// TIA Portal V17 export
// export: Created 2024-03-30T11:15:04.1625877Z, ExportSetting WithDefaults, DisplayName Totally Integrated Automation Portal, DisplayVersion V17, DisplayName TIA Portal Openness, DisplayVersion V17, DisplayName TIA Portal Version Control Interface, DisplayVersion V17, DisplayName STEP 7 Professional, DisplayVersion V17, DisplayName STEP 7 Safety, DisplayVersion V17, DisplayName WinCC Advanced, DisplayVersion V17
TYPE "typ_VGR"
// stored: IsFailsafeCompliant false
   STRUCT
      x_Start_Park_Position : Bool;
      x_Park_Position_Reached : Bool;
      x_NFC_Start_First : Bool;
      x_NFC_Start : Bool;
      x_NFC_Completed : Bool;
      x_HBW_Storage : Bool;
      x_HBW_Outsource : Bool;
      s_HBW_Outsource_Typ : String;
      x_HBW_Discards : Bool;
      x_HBW_PickedUp : Bool;
      x_MPO_Req_Discard : Bool;
      x_MPO_Discards : Bool;
      x_Ready_For_Outsource : Bool;
      x_State_Process : Bool;
      x_Workpiece_NiO : Bool;
      horizontal_Axis : "typ_Axis";
      vertical_Axis : "typ_Axis";
      rotate_Axis : "typ_Axis";
      Workpiece : "typ_Workpiece";
      Worpiece_Parameters { S7_SetPoint := 'True'} : "typ_Workpiece_Parameters";
      History { S7_SetPoint := 'True'} : Array[1..20] of "typ_History";
      di_Pos_DSI_horizontal : DInt;
      di_Pos_DSI_Collect_vertical : DInt;
      di_Pos_DSI_Discard_vertical : DInt;
      di_Offset_Pos_DSI_NFC_vertical : DInt;
      di_Pos_DSI_rotate : DInt;
      di_Pos_DSO_horizontal : DInt;
      di_Pos_DSO_Collect_vertical : DInt;
      di_Pos_DSO_Discard_vertical : DInt;
      di_Offset_Pos_DSO_vertical : DInt;
      di_Pos_DSO_rotate : DInt;
      di_Pos_Color_horizontal : DInt;
      di_Pos_Color_vertical : DInt;
      di_Pos_Color_rotate : DInt;
      di_Pos_NFC_horizontal : DInt;
      di_Pos_NFC_vertical : DInt;
      di_Pos_NFC_rotate : DInt;
      di_Pos_MPO_horizontal : DInt;
      di_Pos_MPO_vertical : DInt;
      di_Offset_Pos_MPO_vertical : DInt;
      di_Pos_MPO_rotate : DInt;
      di_Pos_Free_MPO_Min_rotate : DInt;
      di_Pos_Free_MPO_Max_rotate : DInt;
      di_Pos_Free_MPO_horizontal : DInt;
      di_Pos_HBW_horizontal : DInt;
      di_Offset_Pos_HBW_horizontal : DInt;
      di_Pos_HBW_Collect_vertical : DInt;
      di_Pos_HBW_Discard_vertical : DInt;
      di_Offset_Pos_HBW_vertical : DInt;
      di_Pos_HBW_rotate : DInt;
      di_Pos_NiO_horizontal : DInt;
      di_Pos_NiO_vertical : DInt;
      di_Pos_NiO_rotate : DInt;
      di_Pos_SLD_Blue_horizontal : DInt;
      di_Pos_SLD_Blue_vertical : DInt;
      di_Pos_SLD_Blue_rotate : DInt;
      di_Pos_SLD_Red_horizontal : DInt;
      di_Pos_SLD_Red_vertical : DInt;
      di_Pos_SLD_Red_rotate : DInt;
      di_Pos_SLD_White_horizontal : DInt;
      di_Pos_SLD_White_vertical : DInt;
      di_Pos_SLD_White_rotate : DInt;
      di_Pos_Park_horizontal : DInt;
      di_Pos_Park_vertical : DInt;
      di_Pos_Park_rotate : DInt;
      x_Ready_For_Order : Bool;
   END_STRUCT;
END_TYPE
